{attribute 'qualified_only'}
{attribute 'strict'}
TYPE eLEDSteps :
(
	initialise,	
	running
);
END_TYPE

(* stored: Version 1.1.0.1, ProductVersion 3.1.4026.18
   DUT eLEDSteps: Id {58c43465-10d2-41dd-9ac2-6e2428381179} *)
